FUNCTION_BLOCK btb1
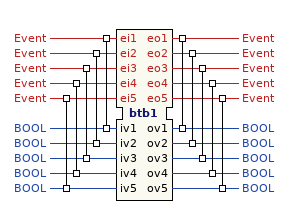
  EVENT_INPUT
    ei1 WITH iv1;
    ei2 WITH iv2;
    ei3 WITH iv3;
    ei4 WITH iv4;
    ei5 WITH iv5;
  END_EVENT
  EVENT_OUTPUT
    eo1 WITH ov1;
    eo2 WITH ov2;
    eo3 WITH ov3;
    eo4 WITH ov4;
    eo5 WITH ov5;
  END_EVENT
  VAR_INPUT
    iv1 : BOOL;
    iv2 : BOOL;
    iv3 : BOOL;
    iv4 : BOOL;
    iv5 : BOOL;
  END_VAR
  VAR_OUTPUT
    ov1 : BOOL;
    ov2 : BOOL;
    ov3 : BOOL;
    ov4 : BOOL;
    ov5 : BOOL;
  END_VAR
  EC_STATES
    START;
  END_STATES
END_FUNCTION_BLOCK
